FUNCTION WRITE_ANY_INT : BOOL
VAR_INPUT
    ptr: POINTER TO INT;
    val: INT;
END_VAR

ptr^ := val;

END_FUNCTION

(* stored: Version 1.1.0.1, ProductVersion 3.1.4022.9
   POU WRITE_ANY_INT: Id {d5d23a20-8f67-4a43-b9e4-bf7852dc7164}, SpecialFunc None *)
